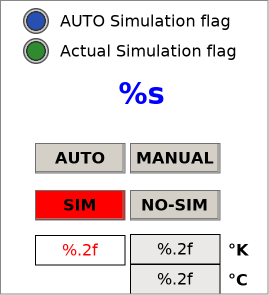
VISUALIZATION GUI_TEMPLATE_TEMP_OVERRIDE  // 269x295
VAR_IN_OUT
	m_Cmd:		FB_CRYO_CMD_OVERRIDE;
	m_Temp:		FB_CRYO_TEMPERATURE;
END_VAR
    Button (35,190 90x30), "SIM", tooltip "Activate Simulation", colour toggle: (m_Cmd.bPermitOn AND NOT m_Cmd.bAutoMode) OR m_Cmd.bEngMode, input disabled if: m_Cmd.bDisableBtnOn
        OnMouseClick: execute { m_Cmd.bManualCmd := TRUE; }
    Lamp1 (21,36 30x30), tooltip "Actual Simulation flag going out", variable: m_Cmd.out_bEnable, style: Lamp-Lamp1-Green
    Rectangle (57,36 200x30), "Actual Simulation flag", tooltip "Actual Simulation flag set the user"
    Button (35,143 90x30), "AUTO", tooltip "Switch to AUTO Mode", colour toggle: m_Cmd.bAutoMode, input disabled if: m_Cmd.bAutoMode OR m_Cmd.bEngMode
        OnMouseClick: execute { m_Cmd.bAutoMode := TRUE; }
    Button (130,143 90x30), "MANUAL", tooltip "Switch to MANUAL Mode", colour toggle: NOT m_Cmd.bAutoMode, input disabled if: NOT m_Cmd.bAutoMode AND NOT m_Cmd.bEngMode
        OnMouseClick: execute { m_Cmd.bAutoMode := FALSE; }
    Button (130,190 90x30), "NO-SIM", tooltip "Deactivate Simulation", colour toggle: (m_Cmd.bPermitOff AND NOT m_Cmd.bAutoMode) OR m_Cmd.bEngMode, input disabled if: m_Cmd.bDisableBtnOff
        OnMouseClick: execute { m_Cmd.bManualCmd := FALSE; }
    Lamp1 (21,6 30x30), tooltip "Simulation flag coming from the Control System", variable: m_Cmd.in_bEnable, style: Lamp-Lamp1-Blue
    Rectangle (57,6 200x30), "AUTO Simulation flag", tooltip "AUTO Simulation flag set by the system"
    Rectangle (67,73 150x41), "%s", text variable: m_Cmd.out_sMode
    Rectangle (35,235 90x30), "%.2f", tooltip "Simulated value [K] when simulation is active.", text variable: m_Temp.stat.lrSimTempK, input disabled if: m_Cmd.bDisableBtnOn OR NOT m_Cmd.out_bEnable
        OnMouseClick: write the text variable via Default
    Rectangle (130,234 90x30), "%.2f", tooltip "Value used by the system [K]", text variable: m_Temp.stat.lrTempK
    Label (225,235 44x30), "°K"
    Rectangle (130,264 90x30), "%.2f", tooltip "Value used by the system [C]", text variable: m_Temp.stat.lrTempC
    Label (225,265 44x30), "°C"
END_VISUALIZATION

(* stored: Version 1.1.0.1, ProductVersion 3.1.4024.12
   Visu GUI_TEMPLATE_TEMP_OVERRIDE: Id {64cc9e6e-3d3e-489b-9561-3881f5a5d25a} *)
